// Visualisaties/OverzetterHMI
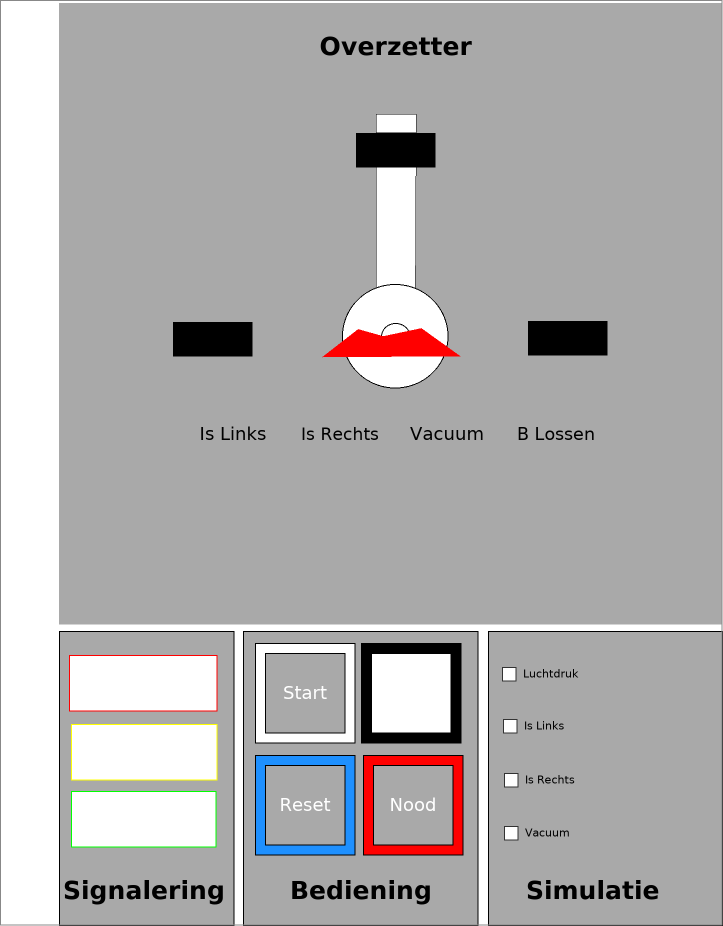
VISUALIZATION OverzetterHMI  // 723x926
    Rectangle (58,2 664x623)
    Polygon (233,394) (233,394) (273,434) (233,474) (193,434), "Is Links", colour toggle: Ix_OverzetterisLinks
    Polygon (340,394) (340,394) (380,434) (340,474) (300,434), "Is Rechts", colour toggle: Ix_OverzetterIsRechts
    Polygon (447,394) (447,394) (487,434) (447,474) (407,434), "Vacuum", colour toggle: Ix_VacuumAanwezig
    Polygon (376,131) (391,131) (416,131) (415,310) (376,310)
        p2858320360: SIM.Vx_OvzRotate
    Polygon (556,394) (556,394) (596,434) (556,474) (516,434), "B Lossen", colour toggle: Qx_BekerLossen
    Polygon (376,114) (391,114) (416,114) (416,132) (376,132), colour toggle: Qx_VacuumAan
        p2858320360: SIM.Vx_OvzRotate
    Polygon (356,133) (371,133) (435,133) (435,167) (356,167), invisible if: SIM.Vx_OvzBlokOverzetter
        p2277200375: SIM.Vx_OvzRotate
    Polygon (173,322) (188,322) (252,322) (252,356) (173,356), invisible if: SIM.Vx_OvzBlokLinks
    Polygon (528,321) (543,321) (607,321) (607,355) (528,355), invisible if: SIM.Vx_OvzBlokRechts
    Ellipse (342,284 106x104)
    Ellipse (381,323 29x27)
    Polygon (358,329) (383,336) (421,328) (460,356) (322,357), invisible if: SIM.Vx_OvzBlokGevallen
        p2277200375: SIM.Vx_OvzRotate
    Label (294,31 204x30), "Overzetter"
    Group (59,631 175x295)
        Rectangle (0,0 175x295)
        Rectangle (10,24 148x56), colour toggle: Qx_RodeLamp
        Rectangle (12,93 146x56), colour toggle: Qx_GeleLamp
        Rectangle (12,160 145x56), colour toggle: Qx_GroeneLamp
        Label (10,236 150x46), "Signalering"
    Group (243,631 235x295)
        Rectangle (0,0 235x295)
        Group (12,12 100x100)
            RoundedRectangle (0,0 100x100)
            RoundedRectangle (10,10 80x80), "Start", tooltip "Start knop", colour toggle: Ix_Startknop
                OnMouseDown: execute { Ix_Startknop := TRUE; }
                OnMouseUp: execute { Ix_Startknop := FALSE; }
        Group (118,12 100x100)
            RoundedRectangle (0,0 100x100)
            RoundedRectangle (10,10 80x80), "Stop", tooltip "Stop knop", colour toggle: Ix_Stopknop
                OnMouseDown: execute { Ix_Stopknop := FALSE; }
                OnMouseUp: execute { Ix_Stopknop := TRUE; }
        Group (12,124 100x100)
            RoundedRectangle (0,0 100x100)
            RoundedRectangle (10,10 80x80), "Reset", tooltip "Reset knop", colour toggle: Ix_Resetknop
                OnMouseDown: execute { Ix_Resetknop := TRUE; }
                OnMouseUp: execute { Ix_Resetknop := FALSE; }
        Group (120,124 100x100)
            RoundedRectangle (0,0 100x100), "Nood"
            RoundedRectangle (10,10 80x80), "Nood", tooltip "Noodstop", colour toggle: Ix_Noodstop
                OnMouseDown: execute { Ix_Noodstop := NOT Ix_Noodstop; }
        Label (43,236 150x46), "Bediening"
    Group (488,631 235x295)
        Group (0,0 235x295)
            Rectangle (0,0 235x295)
            Label (30,236 150x46), "Simulatie"
        Checkbox (12,17 196x52), "Luchtdruk", variable: SIM.Vx_OvzLuchtDrukError
        Checkbox (13,69 196x52), "Is Links", variable: SIM.Vx_OvzIsLinksError
        Checkbox (14,123 196x52), "Is Rechts", variable: SIM.Vx_OvzIsRechtsError
        Checkbox (14,176 196x52), "Vacuum", variable: SIM.Vx_OvzVacuumError
END_VISUALIZATION

// Visualisaties/SorterenHMI
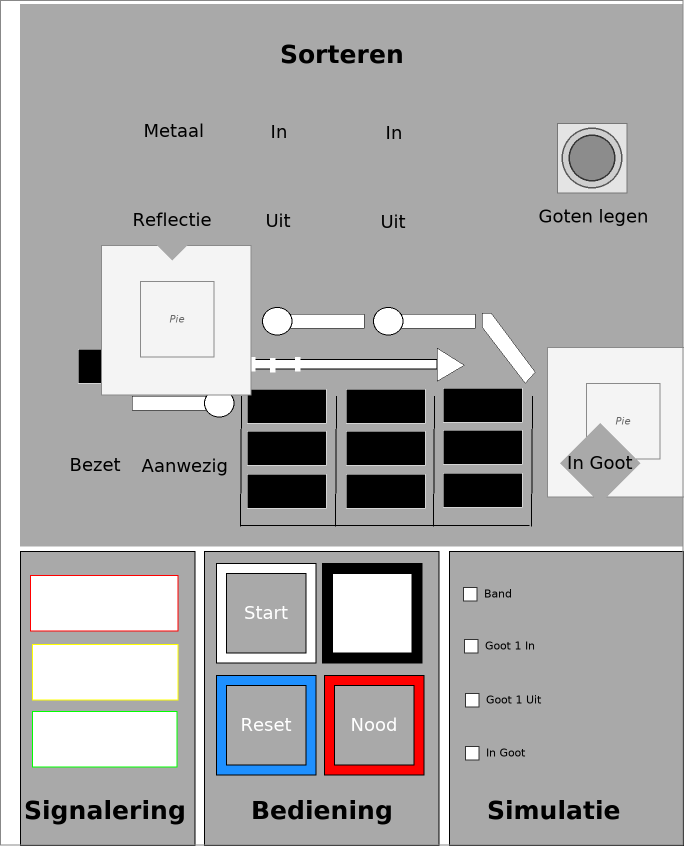
VISUALIZATION SorterenHMI  // 684x846
    Rectangle (19,3 664x544)
    Group (215,348 249x33)
        Rectangle (0,11 222x10), colour toggle: GVL.Qx_MotorAfvoerAan
        Polygon (222,9) (222,0) (249,17) (222,33) (222,22), colour toggle: GVL.Qx_MotorAfvoerAan
        Rectangle (4,9 5x14)
        Rectangle (18,9 5x14)
        Rectangle (35,9 5x14)
        Rectangle (55,10 5x14)
        Rectangle (80,9 5x14)
    Polygon (279,92) (279,92) (319,132) (279,172) (239,132), "In", colour toggle: GVL.Ix_UitvoerGoot1IsIn
    Polygon (278,181) (278,181) (318,221) (278,261) (238,221), "Uit", colour toggle: GVL.Ix_UitvoerGoot1IsUit
    Polygon (78,349) (93,349) (157,349) (157,383) (78,383), invisible if: SIM.Vw_SorBlokBand, colour variable: SIM.Vw_SorKleurBand
        p3560616238: SIM.Vi_SorBlokBandX
        p2738717112: SIM.Vi_SorBlokBandY
    Polygon (247,389) (262,389) (326,389) (326,423) (247,423), invisible if: SIM.Vx_SorBlokGoot[1,1], colour variable: SIM.Vw_SorKleurGoot[1,1]
    Polygon (247,431) (262,431) (326,431) (326,465) (247,465), invisible if: SIM.Vx_SorBlokGoot[1,2], colour variable: SIM.Vw_SorKleurGoot[1,2]
    Polygon (247,474) (262,474) (326,474) (326,508) (247,508), invisible if: SIM.Vx_SorBlokGoot[1,3], colour variable: SIM.Vw_SorKleurGoot[1,3]
    Polygon (346,389) (361,389) (425,389) (425,423) (346,423), invisible if: SIM.Vx_SorBlokGoot[2,1], colour variable: SIM.Vw_SorKleurGoot[2,1]
    Polygon (346,431) (361,431) (425,431) (425,465) (346,465), invisible if: SIM.Vx_SorBlokGoot[2,2], colour variable: SIM.Vw_SorKleurGoot[2,2]
    Polygon (346,474) (361,474) (425,474) (425,508) (346,508), invisible if: SIM.Vx_SorBlokGoot[2,3], colour variable: SIM.Vw_SorKleurGoot[2,3]
    Polygon (443,388) (458,388) (522,388) (522,422) (443,422), invisible if: SIM.Vx_SorBlokGoot[3,1], colour variable: SIM.Vw_SorKleurGoot[3,1]
    Polygon (443,430) (458,430) (522,430) (522,464) (443,464), invisible if: SIM.Vx_SorBlokGoot[3,2], colour variable: SIM.Vw_SorKleurGoot[3,2]
    Polygon (443,473) (458,473) (522,473) (522,507) (443,507), invisible if: SIM.Vx_SorBlokGoot[3,3], colour variable: SIM.Vw_SorKleurGoot[3,3]
    Polygon (132,396) (187,396) (210,396) (210,410) (132,410)
        p2858320360: SIM.Vw_SorStopperRotate
    Ellipse (204,389 30x28)
    Polygon (286,314) (341,314) (364,314) (364,328) (286,328)
        p2858320360: SIM.Vw_SorGoot1Rotate
    Ellipse (262,307 30x28)
    Polygon (397,314) (452,314) (475,314) (475,328) (397,328)
        p2858320360: SIM.Vw_SorGoot2Rotate
    Ellipse (373,307 30x28)
    Polygon (482,313) (491,313) (535,372) (525,383) (482,327)
    Group (101,245 80x82)
        Pie (0,0 150x150)
        Pie (39,36 74x76)
    Line (241,396) (240,526)
    Line (336,396) (335,526)
    Line (434,396) (433,526)
    Line (532,396) (531,526)
    Line (241,525) (529,525)
    Group (547,347 65x105)
        Pie (0,0 150x150)
        Pie (39,36 74x76)
    Polygon (394,93) (394,93) (434,133) (394,173) (354,133), "In", colour toggle: GVL.Ix_UitvoerGoot2IsIn
    Polygon (393,182) (393,182) (433,222) (393,262) (353,222), "Uit", colour toggle: GVL.Ix_UitvoerGoot2IsUit
    Polygon (600,423) (600,423) (640,463) (600,503) (560,463), "In Goot", colour toggle: GVL.Ix_BekerInGoot
    Polygon (95,425) (95,425) (135,465) (95,505) (55,465), "Bezet", colour toggle: GVL.Ix_StationAfvoerVrij
    Polygon (174,91) (174,91) (214,131) (174,171) (134,131), "Metaal", colour toggle: GVL.Ix_BekerMetaal
    Polygon (172,180) (172,180) (212,220) (172,260) (132,220), "Reflectie", colour toggle: GVL.Ix_BekerReflecteerd
    Polygon (190,426) (190,426) (230,466) (190,506) (140,466), "Aanwezig", colour toggle: GVL.Ix_BekerAanwezig
    Label (267,39 150x30), "Sorteren"
    Group (20,551 175x295)
        Rectangle (0,0 175x295)
        Rectangle (10,24 148x56), colour toggle: Qx_RodeLamp
        Rectangle (12,93 146x56), colour toggle: Qx_GeleLamp
        Rectangle (12,160 145x56), colour toggle: Qx_GroeneLamp
        Label (10,236 150x46), "Signalering"
    Group (204,551 235x295)
        Rectangle (0,0 235x295)
        Group (12,12 100x100)
            RoundedRectangle (0,0 100x100)
            RoundedRectangle (10,10 80x80), "Start", tooltip "Start knop", colour toggle: Ix_Startknop
                OnMouseDown: execute { Ix_Startknop := TRUE; }
                OnMouseUp: execute { Ix_Startknop := FALSE; }
        Group (118,12 100x100)
            RoundedRectangle (0,0 100x100)
            RoundedRectangle (10,10 80x80), "Stop", tooltip "Stop knop", colour toggle: Ix_Stopknop
                OnMouseDown: execute { Ix_Stopknop := FALSE; }
                OnMouseUp: execute { Ix_Stopknop := TRUE; }
        Group (12,124 100x100)
            RoundedRectangle (0,0 100x100)
            RoundedRectangle (10,10 80x80), "Reset", tooltip "Reset knop", colour toggle: Ix_Resetknop
                OnMouseDown: execute { Ix_Resetknop := TRUE; }
                OnMouseUp: execute { Ix_Resetknop := FALSE; }
        Group (120,124 100x100)
            RoundedRectangle (0,0 100x100), "Nood"
            RoundedRectangle (10,10 80x80), "Nood", tooltip "Noodstop", colour toggle: Ix_Noodstop
                OnMouseDown: execute { Ix_Noodstop := NOT Ix_Noodstop; }
        Label (43,236 150x46), "Bediening"
    Group (449,551 235x295)
        Group (0,0 235x295)
            Rectangle (0,0 235x295)
            Label (30,236 150x46), "Simulatie"
        Checkbox (12,17 196x52), "Band", variable: SIM.Vx_SorMotorAfvoerError
        Checkbox (13,69 196x52), "Goot 1 In", variable: SIM.Vx_SorGoot1InError
        Checkbox (14,123 196x52), "Goot 1 Uit", variable: SIM.Vx_SorGoot1UitError
        Checkbox (14,176 196x52), "In Goot", variable: SIM.Vx_SorGoot1InError
    PushSwitch (557,123 70x70), tooltip "Goten legen", variable: SIM.Ix_GotenLegen, behaviour: TOGGLE, style: Switch-PushSwitch-Gray
    Polygon (516,204) (546,204) (576,204) (671,218) (571,232), "Goten legen", colour toggle: Ix_MagazijnLeeg
END_VISUALIZATION
